// instrument joints control
FUNCTION_BLOCK FB_BasicInstruControl
VAR_INPUT
END_VAR
VAR_OUTPUT
END_VAR
VAR
	// instrument PID control paramters
	m_instruKp:ARRAY[1..5] OF LREAL:=[4(5),0.0];
	m_instruKd:ARRAY[1..5] OF LREAL:=[4(0.25), 0];
	m_instruKi:ARRAY[1..5] OF LREAL:=[4(10.0),0];
	m_instruKiLimit:ARRAY[1..5] OF LREAL:=[5(50.0)];
	m_instruCtrlLimit:ARRAY[1..5] OF LREAL:=[2(120.0), 3(200.0)];
	
	// gripper force level threshold for variable PID parameter
	m_forceLevelThres : ARRAY[1..3] OF LREAL := [40, 70, 101];
	
	// yaw PID control (when fingers grasp with force)
	m_yawKp:ARRAY[1..3] OF LREAL:=[5, 8, 10];
	m_yawKd:ARRAY[1..3] OF LREAL:=[0.25, 0.4, 0.6];
	m_yawKi:ARRAY[1..3] OF LREAL:=[10.0, 15.0, 20.0];
	m_yawKiLimit:LREAL:=100.0;
	m_yawCtrlLimit:LREAL:=200.0;
	
	// max grip force/current(mA)
	m_maxGripForce:LREAL;
	m_maxGripCurrent:LREAL:=150.0;
	
	// max gripper finger control force/current(mA)
	m_maxGripCtrlForce:LREAL;
	m_maxGripCtrlCurrent:LREAL:=250.0;
	
	// ratio convert motor current to joint troque
	m_currentRatioMotor2Jnt:LREAL;
	
	// PID for instrument joint position
	m_instruJntCtrl:ARRAY[1..5] OF FB_PID;

	// PID for instrument yaw angle 
	m_instruYawCtrl : FB_PID;
	
	// command instrument joint position and velocity
	m_instruCmdJntPos:Vec5d;
	m_instruCmdJntVel:Vec5d;
	
	// current instrument joint position and velocity
	m_instruCurJntPos: Vec5d;
	m_instruCurJntVel:Vec5d;
	
	// grasp force level
	m_graspForceLevel:Lreal :=0;
	
	// instrument joint control torque(when gripper is open)
	m_instruJntCtrlTrq:Vec5d:=[5(0.0)];

	// instrument yaw control torque(when gripper is closed)
	m_instruYawCtrlTrq:LREAL;
		
	// current gripper yaw velocity
	m_instruCurYawVel:LREAL;
	
	// yaw angle error(deg)
	m_yawAngErr : LREAL;
	
	// backlash compensation variables
	m_jntBacklash:ARRAY[1..5] OF LREAL:=[5(0)];
	m_instruLastCmdJntPos:Vec5d;
	
	// grip yaw compensation variables
 	m_gripYawCompAng :LREAL;
 	m_maxGripYawCompAng :LREAL;
	m_lastCmdYawAng:LREAL;
	m_jntMoveStep:LREAL := 0.5*g_deg2Rad;
	
END_VAR

METHOD calcBacklash : BOOL
VAR_IN_OUT CONSTANT
	// instrument joint command position
	i_cmdInstruJntPos :Vec5d;
	
	// command yaw position
	i_cmdYawPos : LREAL;
	
	// slave arm data
	i_slaveArm :FB_SlaveArm;
END_VAR

VAR
	i:INT;
	deltaAng:LREAL;
END_VAR
// backslash compensation
FOR i:=1 TO 4 DO
	// integral compensated backslash angle
	deltaAng:=i_cmdInstruJntPos[i]-m_instruLastCmdJntPos[i];
	IF ABS(deltaAng)>m_jntMoveStep THEN
		m_jntBacklash [i] := m_jntBacklash [i] + m_jntMoveStep*sign(deltaAng);
		m_instruLastCmdJntPos[i] := i_cmdInstruJntPos[i];
	END_IF
END_FOR


// exert grip force 
IF m_graspForceLevel >0  THEN
	
	// clear grip finger backlash
	m_jntBacklash [1]:=0;
	m_jntBacklash [2]:=0;
	
	// determin max compensated angle based on grip force 
	FOR i:=1 TO 4 DO 
		IF m_graspForceLevel<= g_instruGripYawCompForceLevel[i] THEN
			m_maxGripYawCompAng := g_instruGripYawCompAng[i];
			EXIT;
		END_IF
	END_FOR

	// compensate yaw joint angle in case it's driven by force difference between two fingers
	IF m_graspForceLevel > 80 AND  ABS(i_cmdYawPos - m_lastCmdYawAng) > m_jntMoveStep  THEN
		m_jntBacklash [3] := m_jntBacklash [3] -  4*m_jntMoveStep*sign(i_cmdYawPos - m_lastCmdYawAng);
	END_IF
	
	// determin  compensated angle
	IF ABS(i_cmdYawPos - m_lastCmdYawAng) > m_jntMoveStep  THEN
		// determin  compensated yaw  angle
		IF (i_cmdYawPos - m_lastCmdYawAng) * m_gripYawCompAng <= 0 THEN
			m_gripYawCompAng := m_gripYawCompAng + 4*m_jntMoveStep * sign(i_cmdYawPos-m_lastCmdYawAng);
		ELSE
			m_gripYawCompAng := m_gripYawCompAng + 2*m_jntMoveStep * sign(i_cmdYawPos-m_lastCmdYawAng);
		END_IF
		m_lastCmdYawAng := i_cmdYawPos;
	END_IF
	m_gripYawCompAng := LIMIT(-m_maxGripYawCompAng, m_gripYawCompAng,m_maxGripYawCompAng);
	

ELSE
	m_gripYawCompAng:=0;
	m_lastCmdYawAng := i_cmdYawPos;
END_IF

// limit compensated backslash angle
FOR i:=1 TO 4 DO

	IF i<3 THEN 
		IF g_instruBacklashDir[i] > 0 THEN
			m_jntBacklash [i] := LIMIT(0, m_jntBacklash[i], i_slaveArm.instrument.instruTypeInfo.m_instruYawBacklash);		
		ELSE
			m_jntBacklash [i] := LIMIT(-i_slaveArm.instrument.instruTypeInfo.m_instruYawBacklash, m_jntBacklash[i], 0);	
		END_IF

	ELSIF i=3 THEN
		IF g_instruBacklashDir[i] > 0 THEN
			m_jntBacklash [i] := LIMIT(0, m_jntBacklash[i], i_slaveArm.instrument.instruTypeInfo.m_instruPitchBachlash);
		ELSE
			m_jntBacklash [i] := LIMIT(-i_slaveArm.instrument.instruTypeInfo.m_instruPitchBachlash, m_jntBacklash[i], 0);	
		END_IF
	ELSE
		m_jntBacklash [i]:=0;
	END_IF
	
END_FOR
END_METHOD

METHOD PUBLIC clearBacklash : BOOL
VAR_INPUT
END_VAR
m_jntBacklash := g_zeroVec5d;
END_METHOD

METHOD init : BOOL
VAR_IN_OUT CONSTANT
	i_slaveArm:FB_SlaveArm;
END_VAR

VAR
	i,j:INT;
END_VAR
m_graspForceLevel:=0;

// init controller
m_maxGripCurrent:= i_slaveArm.instrument.instruTypeInfo.m_normGripTrq;
m_currentRatioMotor2Jnt:=GVL_SlaveMotorParameters.g_motorTrqConst[4]*GVL_SlaveMotorParameters.g_motorReduction[4]/1000;
m_maxGripForce := m_maxGripCurrent * m_currentRatioMotor2Jnt;
m_maxGripCtrlForce := m_maxGripCtrlCurrent * m_currentRatioMotor2Jnt;
FOR i:=1 TO 4 DO
	m_instruCmdJntPos[i]:=i_slaveArm.curJntPos[i+3];
	
	m_instruCmdJntVel[i]:=0;
	
	m_instruJntCtrl[i].init(g_slaveArmCtrlCycleTime,m_instruKp[i],m_instruKd[i],m_instruKi[i],
		m_instruKiLimit[i]* m_currentRatioMotor2Jnt,	m_instruCtrlLimit[i]*m_currentRatioMotor2Jnt);
	
	m_instruLastCmdJntPos[i]:=m_instruCmdJntPos[i];
END_FOR
m_instruYawCtrl.init(g_slaveArmCtrlCycleTime,m_yawKp[1],m_yawKd[1],m_yawKi[1],m_yawKiLimit*m_currentRatioMotor2Jnt, m_yawCtrlLimit*m_currentRatioMotor2Jnt);
END_METHOD

METHOD run : BOOL
VAR_IN_OUT CONSTANT
	// instrument joint command position
	i_cmdInstruJntPos :Vec5d;
	
	// instrument joint command velocity
	i_cmdInstruJntVel :Vec5d;
	
	// command yaw position
	i_cmdYawPos : LREAL;
	
	// command yaw velocity
	i_cmdYawVel :LREAL;
	
	// command grip force level
	i_cmdGripForceLevel:LREAL;
	
	// slave arm data
	i_slaveArm :FB_SlaveArm;
END_VAR

VAR_OUTPUT
	// joint control torque
	o_cmdJntTrq:Vec5d;
END_VAR

VAR
	i: INT;
	deltaAng:LREAL;
END_VAR
m_graspForceLevel:=LIMIT(0,i_cmdGripForceLevel ,  100)	;

// calculate instrument backlash
calcBacklash(i_cmdInstruJntPos, i_cmdYawPos, i_slaveArm);


// joint position control
FOR i:=1 TO 4 DO	
	m_instruCmdJntPos[i]:=i_cmdInstruJntPos[i];
	m_instruCmdJntVel[i]:=i_cmdInstruJntVel[i];
	m_instruCurJntPos[i]:=i_slaveArm.curJntPos[i+3];
	m_instruCurJntVel[i]:= i_slaveArm.curJntVel[i+3];
	m_instruJntCtrlTrq[i]:=m_instruJntCtrl[i].run(m_instruCmdJntPos[i] ,m_instruCurJntPos[i], m_instruCmdJntVel[i], m_instruCurJntVel[i]);
END_FOR
m_instruJntCtrlTrq[5]:=0;

m_instruCurYawVel :=i_slaveArm.curDHJntVel[6];
m_yawAngErr:=g_rad2Deg*(i_cmdYawPos-i_slaveArm.curDHJntPos[6]);


// exert grip force 
IF m_graspForceLevel >0  THEN
	
	// varialbe PID control based on different gripper force level
	FOR i:=1 TO 3 DO 
		IF m_graspForceLevel < m_forceLevelThres[i] THEN
			m_instruYawCtrl.setPIDParam(m_yawKp[i],m_yawKd[i],m_yawKi[i]);
			EXIT;
		END_IF
	END_FOR

	// yaw control
	m_instruYawCtrlTrq:=m_instruYawCtrl.run(i_cmdYawPos+m_gripYawCompAng,i_slaveArm.curDHJntPos[6],i_cmdYawVel, m_instruCurYawVel);

	// add feed forward grasp force
	m_instruJntCtrlTrq[1]:= m_maxGripForce*m_graspForceLevel/100.0 + m_instruYawCtrlTrq;
	m_instruJntCtrlTrq[2]:= m_maxGripForce*m_graspForceLevel/100.0 - m_instruYawCtrlTrq;
	m_instruJntCtrlTrq[1]:=LIMIT(-m_maxGripForce/10.0,m_instruJntCtrlTrq[1], m_maxGripCtrlForce);
	m_instruJntCtrlTrq[2]:=LIMIT(-m_maxGripForce/10.0,m_instruJntCtrlTrq[2], m_maxGripCtrlForce);
END_IF

o_cmdJntTrq := m_instruJntCtrlTrq;
END_METHOD

METHOD setMaxGripTrq : BOOL
VAR_INPUT
	i_maxGripTrq:LREAL;
END_VAR
m_maxGripCurrent := i_maxGripTrq;
m_maxGripForce := m_maxGripCurrent * m_currentRatioMotor2Jnt;
END_METHOD

END_FUNCTION_BLOCK

(* stored: Version 1.1.0.1, ProductVersion 3.1.4024.12
   POU FB_BasicInstruControl: Id {133d07e3-99c5-4338-ad65-0a5f3241047e}, SpecialFunc None
   Method calcBacklash: Id {32c8ba49-4d3e-4521-a27d-e201d0ada28f}
   Method clearBacklash: Id {be952804-e2b5-49e4-ae4f-cb40af1d0d31}
   Method init: Id {ad68ad31-14f3-42f4-bf27-26d385743fba}
   Method run: Id {7565c7b3-97d9-43dd-bc18-57a80d3fc9eb}
   Method setMaxGripTrq: Id {bb3c440d-4ac6-4283-81ed-1c22dc0afb05} *)
